# EPICS autosave request: ADApp/Db/NDTimeSeries_settingsN.req
# This works for one ROI
$(P)$(R)Name
$(P)$(R)Use
